FUNCTION_BLOCK MOTION_COUNTER_RESET
VAR_INPUT
	BOOL_JOG_ACTIVE : BOOL;
	TIME_RST_DELAY_OFF : TIME;
END_VAR
VAR_OUTPUT
	COUNTER_RST_BOOL : BOOL;
END_VAR
VAR
	DFN: F_TRIG;
	JOGDFN: BOOL;
	T1: TON;
	T1ON: BOOL;
	t0: TON;
	CUTDELAY: BOOL;
END_VAR

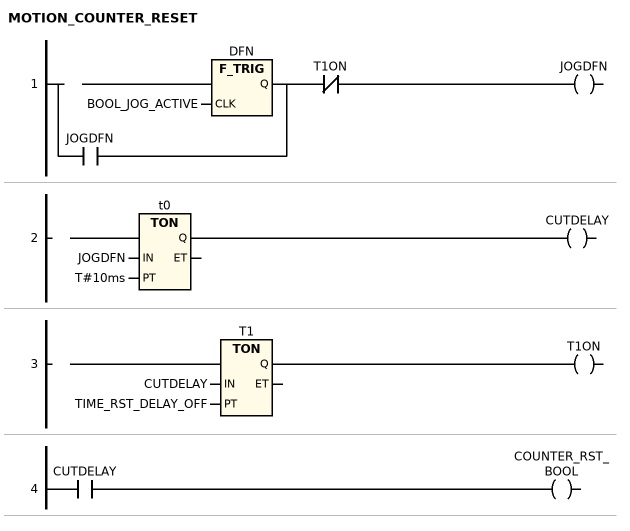
// NETWORK 1
DFN(CLK := BOOL_JOG_ACTIVE); // F_TRIG
JOGDFN := (DFN.Q OR JOGDFN) AND NOT T1ON;

// NETWORK 2
t0(IN := JOGDFN, PT := T#10ms); // TON
CUTDELAY := t0.Q;

// NETWORK 3
T1(IN := CUTDELAY, PT := TIME_RST_DELAY_OFF); // TON
T1ON := T1.Q;

// NETWORK 4
COUNTER_RST_BOOL := CUTDELAY;

END_FUNCTION_BLOCK

(* stored: Version 1.1.0.1, ProductVersion 3.1.4024.12
   POU MOTION_COUNTER_RESET: Id {9637431c-f1a6-42d2-b71c-7dc06ad1984c}, SpecialFunc None *)
